(*
  QualiVision line camera system
  DMAX76.   
*)
FUNCTION_BLOCK FB_LineCamera585 EXTENDS FB_LineCamera

VAR CONSTANT
  cCameraWidth585            : DINT := 9216;     (*Camera width [px]*)
  cCameraMechOffsetTC585     : REAL := 101.5;    (*Camera mechanical offset at calibration temp [mm]*)
  cMechOffsetCameraToPU585   : REAL :=  13.039;  (*Camera mechanical offset to PrintUnit [mm]*)
  cPrintUnitMechOffsetTC585  : REAL :=  32.9869; (*PrintUnit mechanical offset at calibration temp [mm]*)
END_VAR

SUPER^();

METHOD InitLineCamera
VAR_INPUT
  nPrintUnitResolution         : UDINT;    (*printhead pixel resolution [dpi]*)
  nPrintUnitSubPx              : UDINT;    (*print unit subPixel resolution [SubPx]*)
  nPrintUnitWidth              : UDINT;    (*print unit width in [px]*)
  iCameraTrigger               : I_CameraTrigger;
END_VAR
(*Init for dmax type*)
_nCameraWidth           := cCameraWidth585;
_fCameraMechOffsetTC    := cCameraMechOffsetTC585;
_fMechOffsetCameraToPU  := cMechOffsetCameraToPU585;
_fPrintUnitMechOffsetTC := cPrintUnitMechOffsetTC585;

SUPER^.InitLineCamera( nPrintUnitResolution := nPrintUnitResolution
                     , nPrintUnitSubPx      := nPrintUnitSubPx
                     , nPrintUnitWidth      := nPrintUnitWidth
                     , iCameraTrigger       := iCameraTrigger
                     );
END_METHOD

{attribute 'monitoring':='variable'}
PROPERTY sName : STRING
GET
sName := 'LineCam 585';
END_GET
END_PROPERTY

END_FUNCTION_BLOCK

(* stored: Version 1.1.0.1, ProductVersion 3.1.4024.11
   POU FB_LineCamera585: Id {dd79afc7-31bd-4c3b-a5bf-decdb17a1dbd}, SpecialFunc None
   Method InitLineCamera: Id {079361ff-ddae-4fc1-baae-418716f6e04d}
   Property sName: Id {6e1c9c73-2e52-4371-9700-c13bcaafc3f2}
   Get Get: Id {ec506e30-b063-48c2-9272-19fc1383ccfb} *)
